(* PLC project  *)

PROGRAM P
  VAR  (* added by the conversion: wires and edge detectors of the diagram *)
    _ADD3_ENO : BOOL;
    _ADD3_OUT : ANY;
    _MUL6_ENO : BOOL;
    _MUL6_OUT : ANY;
  END_VAR

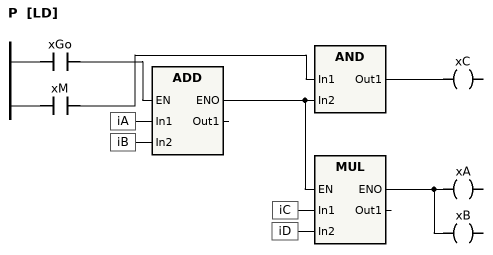
(* LD diagram, written out as Structured Text *)
_ADD3_OUT := ADD(EN := xGo, IN1 := iA, IN2 := iB, ENO => _ADD3_ENO);
_MUL6_OUT := MUL(EN := _ADD3_ENO, IN1 := iC, IN2 := iD, ENO => _MUL6_ENO);
xA := _MUL6_ENO;
xB := _MUL6_ENO;
xC := xM AND _ADD3_ENO;
END_PROGRAM
